// TIA Portal V19 export
TYPE "HU_Pump_Config"
// stored: Access Published
   STRUCT
      SafetyCutOffValveExist : Bool;
      StandbyValveExist : Bool;
      OilPumpContactotFeedbackTimeOut : Time;
   END_STRUCT;
END_TYPE
